Fanuc KAREL source: DISCTRL_ALPH.kl

PROGRAM T
%NOLOCKGROUP
VAR
 v0 : STRING[40]
 v1 : INTEGER
 v2 : INTEGER
 v3 : STRING[40]
 v4 : STRING[40]
 v5 : INTEGER
 v6 : INTEGER
 v7 : INTEGER
BEGIN
 DISCTRL_ALPH(v0, v1, v2, v3, v4, v5, v6, v7)
END T
